FUNCTION IsNone : BOOL
VAR_INPUT
	eResult			: Result;
END_VAR
VAR_OUTPUT
	eCarry			: Result;
END_VAR

IsNone := eResult = 0;
eCarry := eResult;

END_FUNCTION

(* stored: Version 1.1.0.1
   POU IsNone: Id {0669c756-2af9-48b0-9a82-414df9399dbc}, SpecialFunc None *)
